(* CODESYS project versionlib_1202.library
   Author: Filippo Boido
   Placeholder: VersionLib
   Title: VersionLib
   Version: 1.2.0.2
   Company: FactoryAutomation

Project tree, tasks and I/O mapping:
  libraries: Tc2_Standard, * (Beckhoff Automation GmbH); Tc2_System, * (Beckhoff Automation GmbH); Tc3_Module, * (Beckhoff Automation GmbH); VersionLib, * (FactoryAutomation)
  function CheckVersion [ST]
  function GetBuild [ST]
  function GetMajor [ST]
  function GetMinor [ST]
  function GetRevision [ST]
  global variables Version
*)

// Version
{attribute 'qualified_only'}
VAR_GLOBAL CONSTANT
	Major : UINT;
	Minor : UINT;
	Revision : UINT;
	Build : UINT;
END_VAR

// CheckVersion
FUNCTION CheckVersion : BOOL
VAR_INPUT
	Major : UINT;
	Minor : UINT;
	Revision : UINT;
	Build : UINT;
END_VAR
VAR
END_VAR

IF Major = Version.Major
 AND Minor = Version.Minor
 AND Revision = Version.Revision
 AND Build = Version.Build
THEN
	CheckVersion := TRUE;
END_IF

END_FUNCTION

// GetBuild
FUNCTION GetBuild : UINT
VAR_INPUT
END_VAR
VAR
END_VAR

GetBuild := Version.Build;

END_FUNCTION

// GetMajor
FUNCTION GetMajor : UINT
VAR_INPUT
END_VAR
VAR
END_VAR

GetMajor := Version.Major;

END_FUNCTION

// GetMinor
FUNCTION GetMinor : UINT
VAR_INPUT
END_VAR
VAR
END_VAR

GetMinor := Version.Minor;

END_FUNCTION

// GetRevision
FUNCTION GetRevision : UINT
VAR_INPUT
END_VAR
VAR
END_VAR

GetRevision := Version.Revision;

END_FUNCTION
